// TIA Portal V16 export
// export: Created 2022-11-17T11:55:05.4480097Z, ExportSetting WithDefaults, DisplayName Totally Integrated Automation Portal, DisplayVersion V16 Update 6, DisplayName TIA Portal Version Control Interface, DisplayVersion V16 Update 2, DisplayName TIA Portal Openness, DisplayVersion V16 Update 6, DisplayName SINAMICS Startdrive Advanced, DisplayVersion V16 Update 5, DisplayName SINAMICS Startdrive G130, G150, S120, S150, SINAMICS MV, S210, DisplayVersion V16 Update 5, DisplayName SINAMICS Startdrive G110M, G120, G120C, G120D, G120P, G115D, DisplayVersion V16 Update 5, DisplayName STEP 7 Professional, DisplayVersion V16 Update 6, DisplayName STEP 7 Safety, DisplayVersion V16, DisplayName WinCC Advanced, DisplayVersion V16 Update 6
FUNCTION "FC08_SpoolCarriagePos" : Void   // FC8, LAD
TITLE = Spool carriages Helix40/2 positioning
{ S7_Optimized_Access := 'FALSE' }
AUTHOR : Robopac
VERSION : 0.0
// stored: AutoNumber false, IsIECCheckEnabled false, SetENOAutomatically false, UDAEnableTagReadback false
   VAR_TEMP
      Isteresi : Int;
      TempInt : Int;
      Encoder : Int;
      TempDint1 : DInt;
      TempWord : Word;
      TempDint2 : DInt;
   END_VAR
   VAR_TEMP   // added for the SCL form of the ladder/FBD networks
      _w1 : Bool;
      _w2 : Bool;
   END_VAR
BEGIN

REGION Network 1: Reset spool carriage positioning counter (pulse)
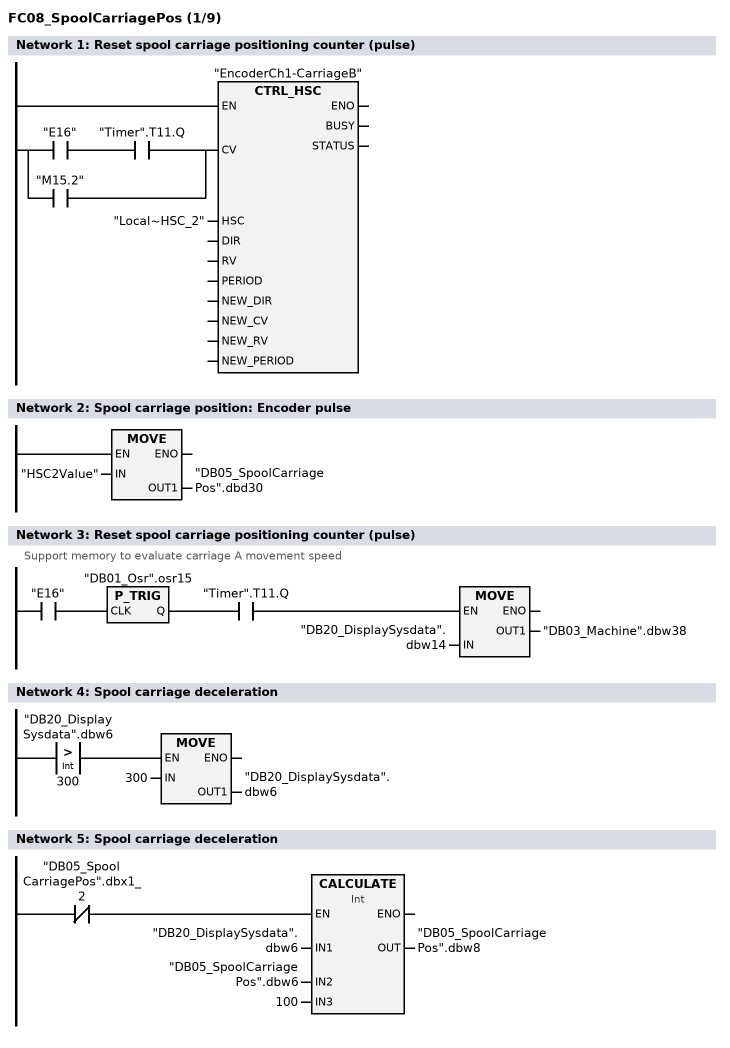
   RUNG wire#powerrail
      "EncoderCh1-CarriageB".CTRL_HSC(CV := wire#w1, HSC := "Local~HSC_2", DIR :=, RV :=, PERIOD :=, NEW_DIR :=, NEW_CV :=, NEW_RV :=, NEW_PERIOD :=, BUSY =>, STATUS =>)
   END_RUNG
   RUNG wire#powerrail
      Contact( "E16" )
      Contact( "Timer".T11.Q )
   END_RUNG wire#w1
   RUNG wire#powerrail
      Contact( "M15.2" )
   END_RUNG wire#w1
   // the same network as SCL:
   "EncoderCh1-CarriageB"(CV := ("E16" AND "Timer".T11.Q) OR "M15.2", HSC := "Local~HSC_2");   // CTRL_HSC
END_REGION

REGION Network 2: Spool carriage position: Encoder pulse
   RUNG wire#powerrail
      { S7_GenerateENO := "TRUE" } Move(in := "HSC2Value", out1 => "DB05_SpoolCarriagePos".dbd30)
   END_RUNG
   // the same network as SCL:
   "DB05_SpoolCarriagePos".dbd30 := "HSC2Value";
END_REGION

REGION Network 3: Reset spool carriage positioning counter (pulse)
   // Support memory to evaluate carriage A movement speed
   RUNG wire#powerrail
      Contact( "E16" )
      P_Trig( "DB01_Osr".osr15 )
      Contact( "Timer".T11.Q )
      { S7_GenerateENO := "TRUE" } Move(in := "DB20_DisplaySysdata".dbw14, out1 => "DB03_Machine".dbw38)
   END_RUNG
   // the same network as SCL:
   #_w1 := "E16" AND NOT "DB01_Osr".osr15;   // rising edge
   "DB01_Osr".osr15 := "E16";
   IF #_w1 AND "Timer".T11.Q THEN "DB03_Machine".dbw38 := "DB20_DisplaySysdata".dbw14; END_IF;
END_REGION

REGION Network 4: Spool carriage deceleration
   RUNG wire#powerrail
      { S7_Templates := "SrcType := Int" } GT_Contact(in1 := "DB20_DisplaySysdata".dbw6, in2 := 300)
      { S7_GenerateENO := "TRUE" } Move(in := 300, out1 => "DB20_DisplaySysdata".dbw6)
   END_RUNG
   // the same network as SCL:
   IF "DB20_DisplaySysdata".dbw6 > 300 THEN "DB20_DisplaySysdata".dbw6 := 300; END_IF;
END_REGION

REGION Network 5: Spool carriage deceleration
   RUNG wire#powerrail
      I_Contact( "DB05_SpoolCarriagePos".dbx1_2 )
      { S7_Templates := "SrcType := Int"; S7_GenerateENO := "TRUE"; S7_Expression := "In1 * In2 / In3" } Calculate(in1 := "DB20_DisplaySysdata".dbw6, in2 := "DB05_SpoolCarriagePos".dbw6, in3 := 100, out => "DB05_SpoolCarriagePos".dbw8)
   END_RUNG
   // the same network as SCL:
   IF NOT "DB05_SpoolCarriagePos".dbx1_2 THEN
       "DB05_SpoolCarriagePos".dbw8 := "DB20_DisplaySysdata".dbw6 * "DB05_SpoolCarriagePos".dbw6 / 100;
   END_IF;
END_REGION

REGION Network 6: Spool carriage position and deceleration
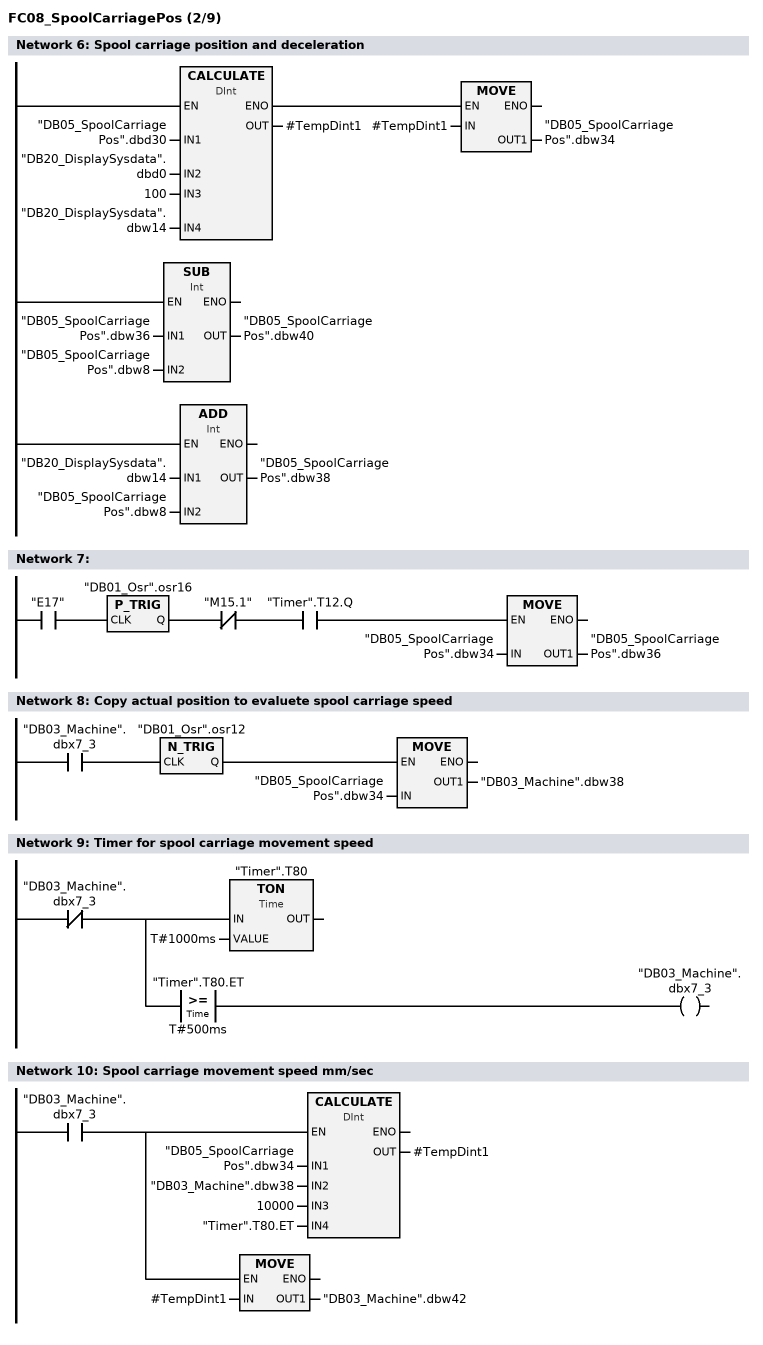
   RUNG wire#powerrail
      { S7_Templates := "SrcType := DInt"; S7_GenerateENO := "TRUE"; S7_Expression := "((In1*In2)/In3)+In4" } Calculate(in1 := "DB05_SpoolCarriagePos".dbd30, in2 := "DB20_DisplaySysdata".dbd0, in3 := 100, in4 := "DB20_DisplaySysdata".dbw14, out => #TempDint1)
      { S7_GenerateENO := "TRUE" } Move(in := #TempDint1, out1 => "DB05_SpoolCarriagePos".dbw34)
   END_RUNG
   RUNG wire#powerrail
      { S7_Templates := "SrcType := Int"; S7_GenerateENO := "TRUE" } Sub(in1 := "DB05_SpoolCarriagePos".dbw36, in2 := "DB05_SpoolCarriagePos".dbw8, out => "DB05_SpoolCarriagePos".dbw40)
   END_RUNG
   RUNG wire#powerrail
      { S7_Templates := "SrcType := Int"; S7_GenerateENO := "TRUE" } Add(in1 := "DB20_DisplaySysdata".dbw14, in2 := "DB05_SpoolCarriagePos".dbw8, out => "DB05_SpoolCarriagePos".dbw38)
   END_RUNG
   // the same network as SCL:
   // ENO of a box is taken as its EN; it also drops when the box reports an error
   #TempDint1 := (("DB05_SpoolCarriagePos".dbd30*"DB20_DisplaySysdata".dbd0)/100)+"DB20_DisplaySysdata".dbw14;
   "DB05_SpoolCarriagePos".dbw34 := #TempDint1;
   "DB05_SpoolCarriagePos".dbw40 := "DB05_SpoolCarriagePos".dbw36 - "DB05_SpoolCarriagePos".dbw8;
   "DB05_SpoolCarriagePos".dbw38 := "DB20_DisplaySysdata".dbw14 + "DB05_SpoolCarriagePos".dbw8;
END_REGION

REGION Network 7
   RUNG wire#powerrail
      Contact( "E17" )
      P_Trig( "DB01_Osr".osr16 )
      I_Contact( "M15.1" )
      Contact( "Timer".T12.Q )
      { S7_GenerateENO := "TRUE" } Move(in := "DB05_SpoolCarriagePos".dbw34, out1 => "DB05_SpoolCarriagePos".dbw36)
   END_RUNG
   // the same network as SCL:
   #_w1 := "E17" AND NOT "DB01_Osr".osr16;   // rising edge
   "DB01_Osr".osr16 := "E17";
   IF #_w1 AND NOT "M15.1" AND "Timer".T12.Q THEN
       "DB05_SpoolCarriagePos".dbw36 := "DB05_SpoolCarriagePos".dbw34;
   END_IF;
END_REGION

REGION Network 8: Copy actual position to evaluete spool carriage speed
   RUNG wire#powerrail
      Contact( "DB03_Machine".dbx7_3 )
      N_Trig( "DB01_Osr".osr12 )
      { S7_GenerateENO := "TRUE" } Move(in := "DB05_SpoolCarriagePos".dbw34, out1 => "DB03_Machine".dbw38)
   END_RUNG
   // the same network as SCL:
   #_w1 := NOT "DB03_Machine".dbx7_3 AND "DB01_Osr".osr12;   // falling edge
   "DB01_Osr".osr12 := "DB03_Machine".dbx7_3;
   IF #_w1 THEN "DB03_Machine".dbw38 := "DB05_SpoolCarriagePos".dbw34; END_IF;
END_REGION

REGION Network 9: Timer for spool carriage movement speed
   #_w1 := NOT "DB03_Machine".dbx7_3;
   "Timer".T80.TON(IN := #_w1, PT := T#1000ms);   // TON coil
   "DB03_Machine".dbx7_3 := #_w1 AND ("Timer".T80.ET >= T#500ms);
END_REGION

REGION Network 10: Spool carriage movement speed mm/sec
   RUNG wire#powerrail
      Contact( "DB03_Machine".dbx7_3 )
      wire#w1
      { S7_Templates := "SrcType := DInt"; S7_GenerateENO := "TRUE"; S7_Expression := "(In1-In2)*In3/In4" } Calculate(in1 := "DB05_SpoolCarriagePos".dbw34, in2 := "DB03_Machine".dbw38, in3 := 10000, in4 := "Timer".T80.ET, out => #TempDint1)
   END_RUNG
   RUNG wire#w1
      { S7_GenerateENO := "TRUE" } Move(in := #TempDint1, out1 => "DB03_Machine".dbw42)
   END_RUNG
   // the same network as SCL:
   IF "DB03_Machine".dbx7_3 THEN
       #TempDint1 := ("DB05_SpoolCarriagePos".dbw34-"DB03_Machine".dbw38)*10000/"Timer".T80.ET;
       "DB03_Machine".dbw42 := #TempDint1;
   END_IF;
END_REGION

REGION Network 11: Spool carriage movement speed mm/sec recorded
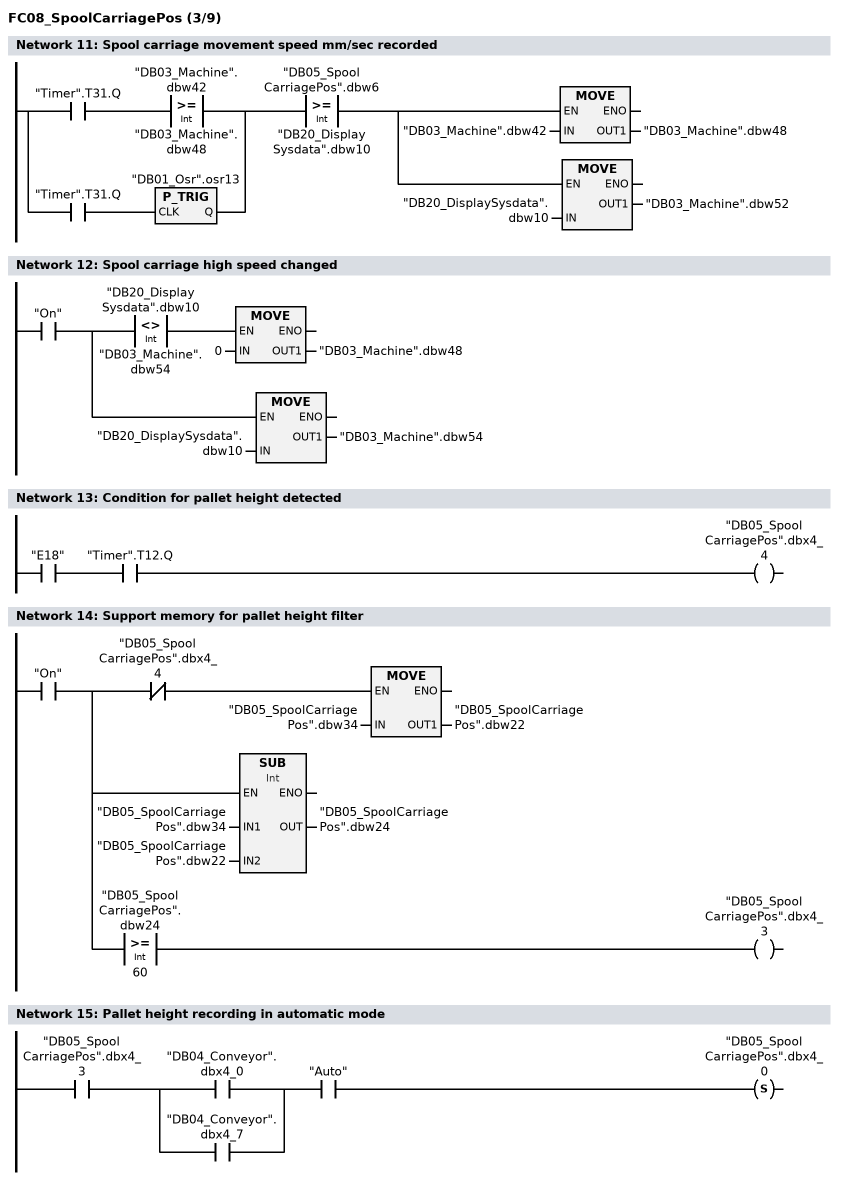
   RUNG wire#powerrail
      Contact( "Timer".T31.Q )
      { S7_Templates := "SrcType := Int" } GE_Contact(in1 := "DB03_Machine".dbw42, in2 := "DB03_Machine".dbw48)
      wire#w1
      { S7_Templates := "SrcType := Int" } GE_Contact(in1 := "DB05_SpoolCarriagePos".dbw6, in2 := "DB20_DisplaySysdata".dbw10)
      wire#w2
      { S7_GenerateENO := "TRUE" } Move(in := "DB03_Machine".dbw42, out1 => "DB03_Machine".dbw48)
   END_RUNG
   RUNG wire#powerrail
      Contact( "Timer".T31.Q )
      P_Trig( "DB01_Osr".osr13 )
   END_RUNG wire#w1
   RUNG wire#w2
      { S7_GenerateENO := "TRUE" } Move(in := "DB20_DisplaySysdata".dbw10, out1 => "DB03_Machine".dbw52)
   END_RUNG
   // the same network as SCL:
   #_w1 := "Timer".T31.Q AND NOT "DB01_Osr".osr13;   // rising edge
   "DB01_Osr".osr13 := "Timer".T31.Q;
   #_w2 := (("Timer".T31.Q AND ("DB03_Machine".dbw42 >= "DB03_Machine".dbw48)) OR #_w1) AND ("DB05_SpoolCarriagePos".dbw6 >= "DB20_DisplaySysdata".dbw10);
   IF #_w2 THEN
       "DB03_Machine".dbw48 := "DB03_Machine".dbw42;
       "DB03_Machine".dbw52 := "DB20_DisplaySysdata".dbw10;
   END_IF;
END_REGION

REGION Network 12: Spool carriage high speed changed
   RUNG wire#powerrail
      Contact( "On" )
      wire#w1
      { S7_Templates := "SrcType := Int" } NE_Contact(in1 := "DB20_DisplaySysdata".dbw10, in2 := "DB03_Machine".dbw54)
      { S7_GenerateENO := "TRUE" } Move(in := 0, out1 => "DB03_Machine".dbw48)
   END_RUNG
   RUNG wire#w1
      { S7_GenerateENO := "TRUE" } Move(in := "DB20_DisplaySysdata".dbw10, out1 => "DB03_Machine".dbw54)
   END_RUNG
   // the same network as SCL:
   IF "On" AND ("DB20_DisplaySysdata".dbw10 <> "DB03_Machine".dbw54) THEN "DB03_Machine".dbw48 := 0; END_IF;
   IF "On" THEN "DB03_Machine".dbw54 := "DB20_DisplaySysdata".dbw10; END_IF;
END_REGION

REGION Network 13: Condition for pallet height detected
   RUNG wire#powerrail
      Contact( "E18" )
      Contact( "Timer".T12.Q )
      Coil( "DB05_SpoolCarriagePos".dbx4_4 )
   END_RUNG
   // the same network as SCL:
   "DB05_SpoolCarriagePos".dbx4_4 := "E18" AND "Timer".T12.Q;
END_REGION

REGION Network 14: Support memory for pallet height filter
   RUNG wire#powerrail
      Contact( "On" )
      wire#w1
      I_Contact( "DB05_SpoolCarriagePos".dbx4_4 )
      { S7_GenerateENO := "TRUE" } Move(in := "DB05_SpoolCarriagePos".dbw34, out1 => "DB05_SpoolCarriagePos".dbw22)
   END_RUNG
   RUNG wire#w1
      { S7_Templates := "SrcType := Int"; S7_GenerateENO := "TRUE" } Sub(in1 := "DB05_SpoolCarriagePos".dbw34, in2 := "DB05_SpoolCarriagePos".dbw22, out => "DB05_SpoolCarriagePos".dbw24)
   END_RUNG
   RUNG wire#w1
      { S7_Templates := "SrcType := Int" } GE_Contact(in1 := "DB05_SpoolCarriagePos".dbw24, in2 := 60)
      Coil( "DB05_SpoolCarriagePos".dbx4_3 )
   END_RUNG
   // the same network as SCL:
   IF "On" AND NOT "DB05_SpoolCarriagePos".dbx4_4 THEN
       "DB05_SpoolCarriagePos".dbw22 := "DB05_SpoolCarriagePos".dbw34;
   END_IF;
   IF "On" THEN
       "DB05_SpoolCarriagePos".dbw24 := "DB05_SpoolCarriagePos".dbw34 - "DB05_SpoolCarriagePos".dbw22;
   END_IF;
   "DB05_SpoolCarriagePos".dbx4_3 := "On" AND ("DB05_SpoolCarriagePos".dbw24 >= 60);
END_REGION

REGION Network 15: Pallet height recording in automatic mode
   RUNG wire#powerrail
      Contact( "DB05_SpoolCarriagePos".dbx4_3 )
      wire#w1
      Contact( "DB04_Conveyor".dbx4_0 )
      wire#w2
      Contact( "Auto" )
      S_Coil( "DB05_SpoolCarriagePos".dbx4_0 )
   END_RUNG
   RUNG wire#w1
      Contact( "DB04_Conveyor".dbx4_7 )
   END_RUNG wire#w2
   // the same network as SCL:
   IF "DB05_SpoolCarriagePos".dbx4_3 AND ("DB04_Conveyor".dbx4_0 OR "DB04_Conveyor".dbx4_7) AND "Auto" THEN
       "DB05_SpoolCarriagePos".dbx4_0 := TRUE;
   END_IF;
END_REGION

REGION Network 16: Recording pallet height for wrapping position
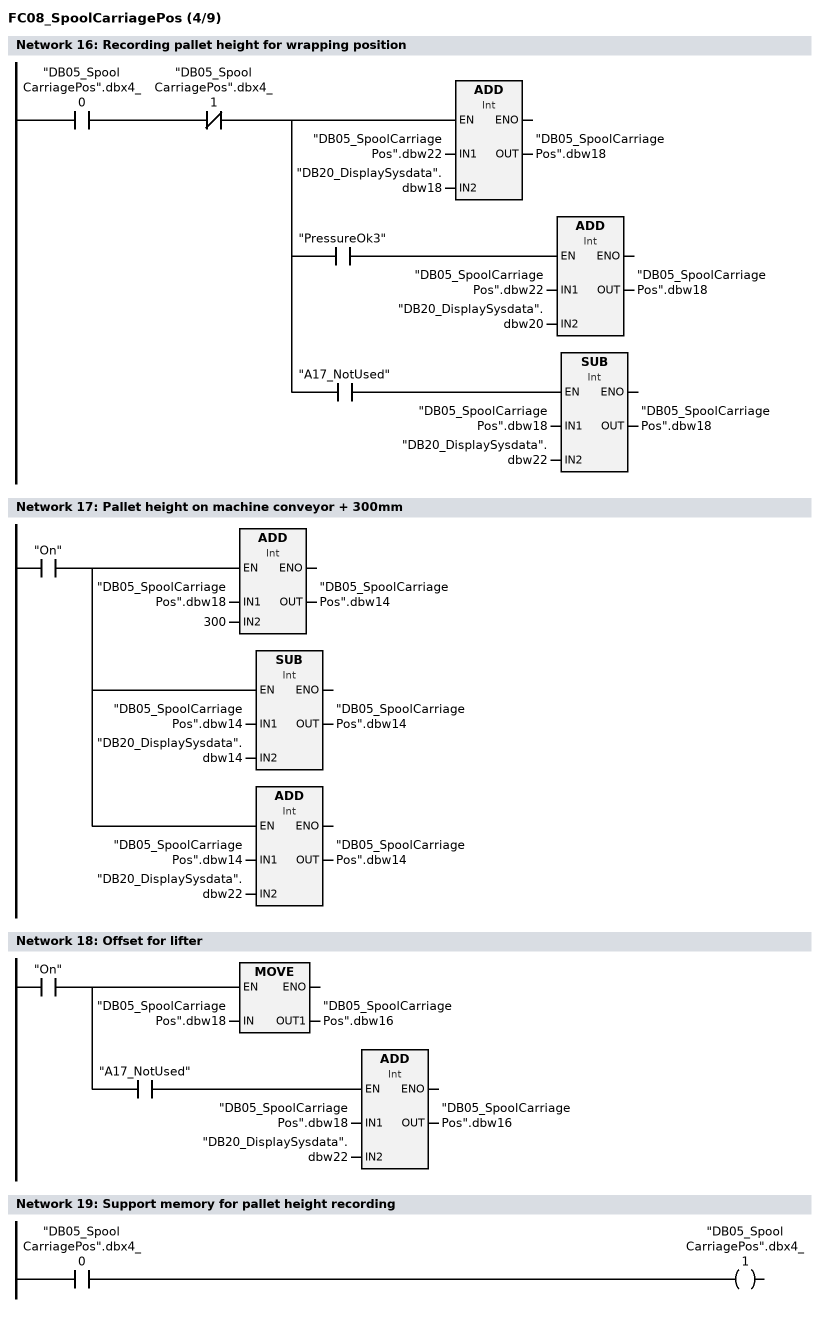
   RUNG wire#powerrail
      Contact( "DB05_SpoolCarriagePos".dbx4_0 )
      I_Contact( "DB05_SpoolCarriagePos".dbx4_1 )
      wire#w1
      { S7_Templates := "SrcType := Int"; S7_GenerateENO := "TRUE" } Add(in1 := "DB05_SpoolCarriagePos".dbw22, in2 := "DB20_DisplaySysdata".dbw18, out => "DB05_SpoolCarriagePos".dbw18)
   END_RUNG
   RUNG wire#w1
      Contact( "PressureOk3" )
      { S7_Templates := "SrcType := Int"; S7_GenerateENO := "TRUE" } Add(in1 := "DB05_SpoolCarriagePos".dbw22, in2 := "DB20_DisplaySysdata".dbw20, out => "DB05_SpoolCarriagePos".dbw18)
   END_RUNG
   RUNG wire#w1
      Contact( "A17_NotUsed" )
      { S7_Templates := "SrcType := Int"; S7_GenerateENO := "TRUE" } Sub(in1 := "DB05_SpoolCarriagePos".dbw18, in2 := "DB20_DisplaySysdata".dbw22, out => "DB05_SpoolCarriagePos".dbw18)
   END_RUNG
   // the same network as SCL:
   #_w1 := "DB05_SpoolCarriagePos".dbx4_0 AND NOT "DB05_SpoolCarriagePos".dbx4_1;
   IF #_w1 THEN
       "DB05_SpoolCarriagePos".dbw18 := "DB05_SpoolCarriagePos".dbw22 + "DB20_DisplaySysdata".dbw18;
   END_IF;
   IF #_w1 AND "PressureOk3" THEN
       "DB05_SpoolCarriagePos".dbw18 := "DB05_SpoolCarriagePos".dbw22 + "DB20_DisplaySysdata".dbw20;
   END_IF;
   IF #_w1 AND "A17_NotUsed" THEN
       "DB05_SpoolCarriagePos".dbw18 := "DB05_SpoolCarriagePos".dbw18 - "DB20_DisplaySysdata".dbw22;
   END_IF;
END_REGION

REGION Network 17: Pallet height on machine conveyor + 300mm
   RUNG wire#powerrail
      Contact( "On" )
      wire#w1
      { S7_Templates := "SrcType := Int"; S7_GenerateENO := "TRUE" } Add(in1 := "DB05_SpoolCarriagePos".dbw18, in2 := 300, out => "DB05_SpoolCarriagePos".dbw14)
   END_RUNG
   RUNG wire#w1
      { S7_Templates := "SrcType := Int"; S7_GenerateENO := "TRUE" } Sub(in1 := "DB05_SpoolCarriagePos".dbw14, in2 := "DB20_DisplaySysdata".dbw14, out => "DB05_SpoolCarriagePos".dbw14)
   END_RUNG
   RUNG wire#w1
      { S7_Templates := "SrcType := Int"; S7_GenerateENO := "TRUE" } Add(in1 := "DB05_SpoolCarriagePos".dbw14, in2 := "DB20_DisplaySysdata".dbw22, out => "DB05_SpoolCarriagePos".dbw14)
   END_RUNG
   // the same network as SCL:
   IF "On" THEN
       "DB05_SpoolCarriagePos".dbw14 := "DB05_SpoolCarriagePos".dbw18 + 300;
       "DB05_SpoolCarriagePos".dbw14 := "DB05_SpoolCarriagePos".dbw14 - "DB20_DisplaySysdata".dbw14;
       "DB05_SpoolCarriagePos".dbw14 := "DB05_SpoolCarriagePos".dbw14 + "DB20_DisplaySysdata".dbw22;
   END_IF;
END_REGION

REGION Network 18: Offset for lifter
   RUNG wire#powerrail
      Contact( "On" )
      wire#w1
      { S7_GenerateENO := "TRUE" } Move(in := "DB05_SpoolCarriagePos".dbw18, out1 => "DB05_SpoolCarriagePos".dbw16)
   END_RUNG
   RUNG wire#w1
      Contact( "A17_NotUsed" )
      { S7_Templates := "SrcType := Int"; S7_GenerateENO := "TRUE" } Add(in1 := "DB05_SpoolCarriagePos".dbw18, in2 := "DB20_DisplaySysdata".dbw22, out => "DB05_SpoolCarriagePos".dbw16)
   END_RUNG
   // the same network as SCL:
   IF "On" THEN "DB05_SpoolCarriagePos".dbw16 := "DB05_SpoolCarriagePos".dbw18; END_IF;
   IF "On" AND "A17_NotUsed" THEN
       "DB05_SpoolCarriagePos".dbw16 := "DB05_SpoolCarriagePos".dbw18 + "DB20_DisplaySysdata".dbw22;
   END_IF;
END_REGION

REGION Network 19: Support memory for pallet height recording
   RUNG wire#powerrail
      Contact( "DB05_SpoolCarriagePos".dbx4_0 )
      Coil( "DB05_SpoolCarriagePos".dbx4_1 )
   END_RUNG
   // the same network as SCL:
   "DB05_SpoolCarriagePos".dbx4_1 := "DB05_SpoolCarriagePos".dbx4_0;
END_REGION

REGION Network 20: Pallet height recording in automatic mode
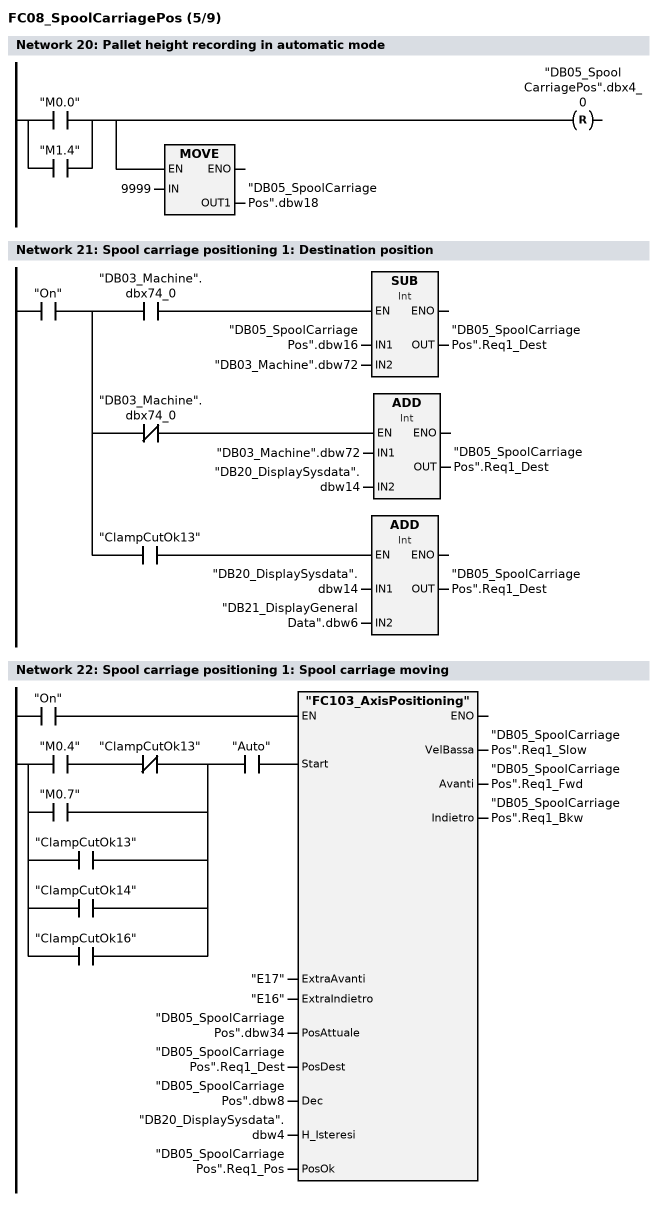
   RUNG wire#powerrail
      Contact( "M0.0" )
      wire#w1
      R_Coil( "DB05_SpoolCarriagePos".dbx4_0 )
   END_RUNG
   RUNG wire#powerrail
      Contact( "M1.4" )
   END_RUNG wire#w1
   RUNG wire#w1
      { S7_GenerateENO := "TRUE" } Move(in := 9999, out1 => "DB05_SpoolCarriagePos".dbw18)
   END_RUNG
   // the same network as SCL:
   IF "M0.0" OR "M1.4" THEN
       "DB05_SpoolCarriagePos".dbx4_0 := FALSE;
       "DB05_SpoolCarriagePos".dbw18 := 9999;
   END_IF;
END_REGION

REGION Network 21: Spool carriage positioning 1: Destination position
   RUNG wire#powerrail
      Contact( "On" )
      wire#w1
      Contact( "DB03_Machine".dbx74_0 )
      { S7_Templates := "SrcType := Int"; S7_GenerateENO := "TRUE" } Sub(in1 := "DB05_SpoolCarriagePos".dbw16, in2 := "DB03_Machine".dbw72, out => "DB05_SpoolCarriagePos".Req1_Dest)
   END_RUNG
   RUNG wire#w1
      I_Contact( "DB03_Machine".dbx74_0 )
      { S7_Templates := "SrcType := Int"; S7_GenerateENO := "TRUE" } Add(in1 := "DB03_Machine".dbw72, in2 := "DB20_DisplaySysdata".dbw14, out => "DB05_SpoolCarriagePos".Req1_Dest)
   END_RUNG
   RUNG wire#w1
      Contact( "ClampCutOk13" )
      { S7_Templates := "SrcType := Int"; S7_GenerateENO := "TRUE" } Add(in1 := "DB20_DisplaySysdata".dbw14, in2 := "DB21_DisplayGeneralData".dbw6, out => "DB05_SpoolCarriagePos".Req1_Dest)
   END_RUNG
   // the same network as SCL:
   IF "On" AND "DB03_Machine".dbx74_0 THEN
       "DB05_SpoolCarriagePos".Req1_Dest := "DB05_SpoolCarriagePos".dbw16 - "DB03_Machine".dbw72;
   END_IF;
   IF "On" AND NOT "DB03_Machine".dbx74_0 THEN
       "DB05_SpoolCarriagePos".Req1_Dest := "DB03_Machine".dbw72 + "DB20_DisplaySysdata".dbw14;
   END_IF;
   IF "On" AND "ClampCutOk13" THEN
       "DB05_SpoolCarriagePos".Req1_Dest := "DB20_DisplaySysdata".dbw14 + "DB21_DisplayGeneralData".dbw6;
   END_IF;
END_REGION

REGION Network 22: Spool carriage positioning 1: Spool carriage moving
   RUNG wire#powerrail
      Contact( "On" )
      "FC103_AxisPositioning"(Start := wire#w2, ExtraAvanti := "E17", ExtraIndietro := "E16", PosAttuale := "DB05_SpoolCarriagePos".dbw34, PosDest := "DB05_SpoolCarriagePos".Req1_Dest, Dec := "DB05_SpoolCarriagePos".dbw8, H_Isteresi := "DB20_DisplaySysdata".dbw4, PosOk := "DB05_SpoolCarriagePos".Req1_Pos, VelBassa => "DB05_SpoolCarriagePos".Req1_Slow, Avanti => "DB05_SpoolCarriagePos".Req1_Fwd, Indietro => "DB05_SpoolCarriagePos".Req1_Bkw)
   END_RUNG
   RUNG wire#powerrail
      Contact( "M0.4" )
      I_Contact( "ClampCutOk13" )
      wire#w1
      Contact( "Auto" )
   END_RUNG wire#w2
   RUNG wire#powerrail
      Contact( "M0.7" )
   END_RUNG wire#w1
   RUNG wire#powerrail
      Contact( "ClampCutOk13" )
   END_RUNG wire#w1
   RUNG wire#powerrail
      Contact( "ClampCutOk14" )
   END_RUNG wire#w1
   RUNG wire#powerrail
      Contact( "ClampCutOk16" )
   END_RUNG wire#w1
   // the same network as SCL:
   IF "On" THEN
       "FC103_AxisPositioning"(Start := (("M0.4" AND NOT "ClampCutOk13") OR "M0.7" OR "ClampCutOk13" OR "ClampCutOk14" OR "ClampCutOk16") AND "Auto",
                               ExtraAvanti := "E17",
                               ExtraIndietro := "E16",
                               PosAttuale := "DB05_SpoolCarriagePos".dbw34,
                               PosDest := "DB05_SpoolCarriagePos".Req1_Dest,
                               Dec := "DB05_SpoolCarriagePos".dbw8,
                               H_Isteresi := "DB20_DisplaySysdata".dbw4,
                               PosOk := "DB05_SpoolCarriagePos".Req1_Pos,
                               VelBassa => "DB05_SpoolCarriagePos".Req1_Slow,
                               Avanti => "DB05_SpoolCarriagePos".Req1_Fwd,
                               Indietro => "DB05_SpoolCarriagePos".Req1_Bkw);
   END_IF;
END_REGION

REGION Network 23: Spool carriage positioning 2: Destination position
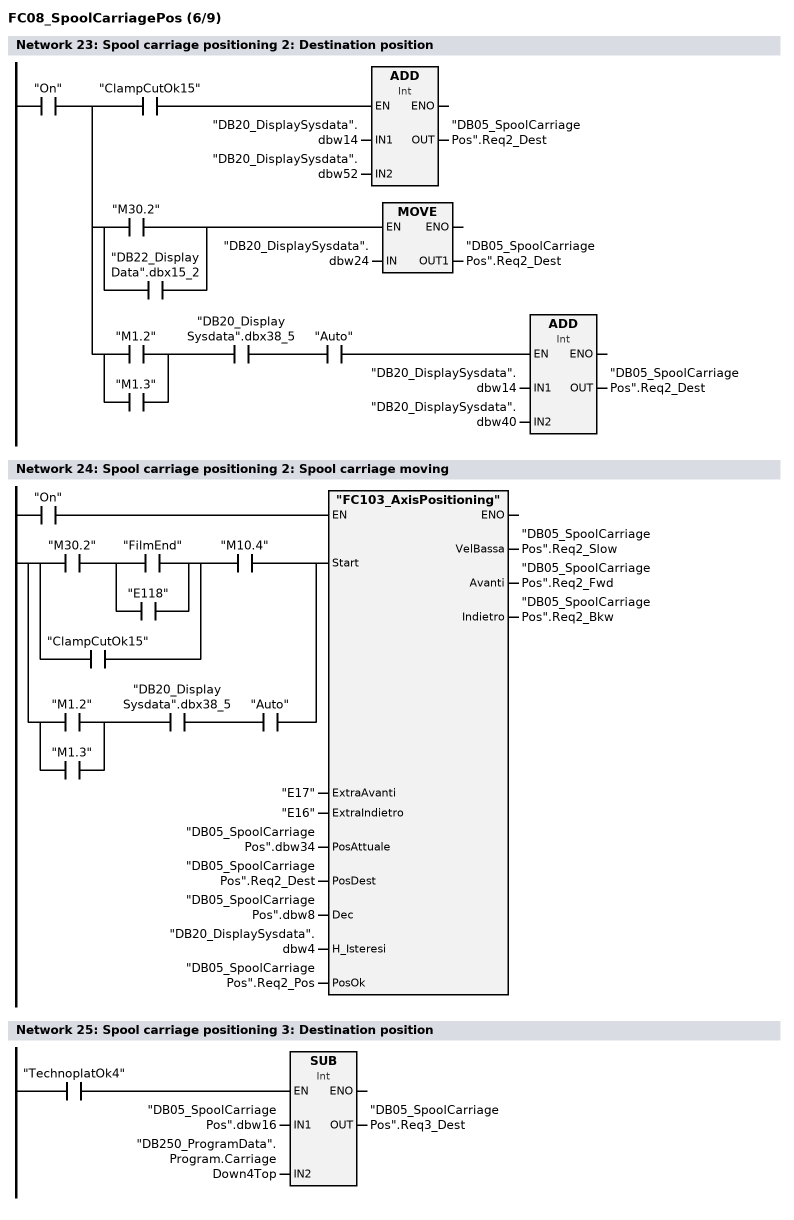
   RUNG wire#powerrail
      Contact( "On" )
      wire#w1
      Contact( "ClampCutOk15" )
      { S7_Templates := "SrcType := Int"; S7_GenerateENO := "TRUE" } Add(in1 := "DB20_DisplaySysdata".dbw14, in2 := "DB20_DisplaySysdata".dbw52, out => "DB05_SpoolCarriagePos".Req2_Dest)
   END_RUNG
   RUNG wire#w1
      Contact( "M30.2" )
      wire#w2
      { S7_GenerateENO := "TRUE" } Move(in := "DB20_DisplaySysdata".dbw24, out1 => "DB05_SpoolCarriagePos".Req2_Dest)
   END_RUNG
   RUNG wire#w1
      Contact( "DB22_DisplayData".dbx15_2 )
   END_RUNG wire#w2
   RUNG wire#w1
      Contact( "M1.2" )
      wire#w3
      Contact( "DB20_DisplaySysdata".dbx38_5 )
      Contact( "Auto" )
      { S7_Templates := "SrcType := Int"; S7_GenerateENO := "TRUE" } Add(in1 := "DB20_DisplaySysdata".dbw14, in2 := "DB20_DisplaySysdata".dbw40, out => "DB05_SpoolCarriagePos".Req2_Dest)
   END_RUNG
   RUNG wire#w1
      Contact( "M1.3" )
   END_RUNG wire#w3
   // the same network as SCL:
   IF "On" AND "ClampCutOk15" THEN
       "DB05_SpoolCarriagePos".Req2_Dest := "DB20_DisplaySysdata".dbw14 + "DB20_DisplaySysdata".dbw52;
   END_IF;
   IF "On" AND ("M30.2" OR "DB22_DisplayData".dbx15_2) THEN
       "DB05_SpoolCarriagePos".Req2_Dest := "DB20_DisplaySysdata".dbw24;
   END_IF;
   IF "On" AND ("M1.2" OR "M1.3") AND "DB20_DisplaySysdata".dbx38_5 AND "Auto" THEN
       "DB05_SpoolCarriagePos".Req2_Dest := "DB20_DisplaySysdata".dbw14 + "DB20_DisplaySysdata".dbw40;
   END_IF;
END_REGION

REGION Network 24: Spool carriage positioning 2: Spool carriage moving
   RUNG wire#powerrail
      Contact( "On" )
      "FC103_AxisPositioning"(Start := wire#w4, ExtraAvanti := "E17", ExtraIndietro := "E16", PosAttuale := "DB05_SpoolCarriagePos".dbw34, PosDest := "DB05_SpoolCarriagePos".Req2_Dest, Dec := "DB05_SpoolCarriagePos".dbw8, H_Isteresi := "DB20_DisplaySysdata".dbw4, PosOk := "DB05_SpoolCarriagePos".Req2_Pos, VelBassa => "DB05_SpoolCarriagePos".Req2_Slow, Avanti => "DB05_SpoolCarriagePos".Req2_Fwd, Indietro => "DB05_SpoolCarriagePos".Req2_Bkw)
   END_RUNG
   RUNG wire#powerrail
      Contact( "M30.2" )
      wire#w1
      Contact( "FilmEnd" )
      wire#w2
      Contact( "M10.4" )
   END_RUNG wire#w4
   RUNG wire#w1
      Contact( "E118" )
   END_RUNG wire#w2
   RUNG wire#powerrail
      Contact( "ClampCutOk15" )
   END_RUNG wire#w2
   RUNG wire#powerrail
      Contact( "M1.2" )
      wire#w3
      Contact( "DB20_DisplaySysdata".dbx38_5 )
      Contact( "Auto" )
   END_RUNG wire#w4
   RUNG wire#powerrail
      Contact( "M1.3" )
   END_RUNG wire#w3
   // the same network as SCL:
   IF "On" THEN
       "FC103_AxisPositioning"(Start := ((("M30.2" AND ("FilmEnd" OR "E118")) OR "ClampCutOk15") AND "M10.4") OR (("M1.2" OR "M1.3") AND "DB20_DisplaySysdata".dbx38_5 AND "Auto"),
                               ExtraAvanti := "E17",
                               ExtraIndietro := "E16",
                               PosAttuale := "DB05_SpoolCarriagePos".dbw34,
                               PosDest := "DB05_SpoolCarriagePos".Req2_Dest,
                               Dec := "DB05_SpoolCarriagePos".dbw8,
                               H_Isteresi := "DB20_DisplaySysdata".dbw4,
                               PosOk := "DB05_SpoolCarriagePos".Req2_Pos,
                               VelBassa => "DB05_SpoolCarriagePos".Req2_Slow,
                               Avanti => "DB05_SpoolCarriagePos".Req2_Fwd,
                               Indietro => "DB05_SpoolCarriagePos".Req2_Bkw);
   END_IF;
END_REGION

REGION Network 25: Spool carriage positioning 3: Destination position
   RUNG wire#powerrail
      Contact( "TechnoplatOk4" )
      { S7_Templates := "SrcType := Int"; S7_GenerateENO := "TRUE" } Sub(in1 := "DB05_SpoolCarriagePos".dbw16, in2 := "DB250_ProgramData".Program.CarriageDown4Top, out => "DB05_SpoolCarriagePos".Req3_Dest)
   END_RUNG
   // the same network as SCL:
   IF "TechnoplatOk4" THEN
       "DB05_SpoolCarriagePos".Req3_Dest := "DB05_SpoolCarriagePos".dbw16 - "DB250_ProgramData".Program.CarriageDown4Top;
   END_IF;
END_REGION

REGION Network 26: Spool carriage positioning 3: Spool carriage moving
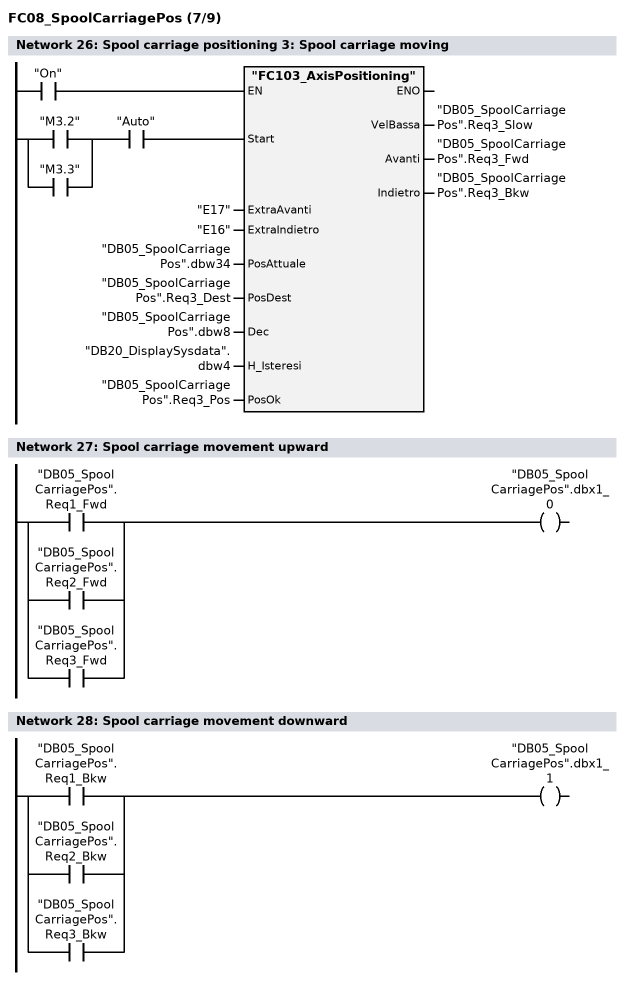
   RUNG wire#powerrail
      Contact( "On" )
      "FC103_AxisPositioning"(Start := wire#w2, ExtraAvanti := "E17", ExtraIndietro := "E16", PosAttuale := "DB05_SpoolCarriagePos".dbw34, PosDest := "DB05_SpoolCarriagePos".Req3_Dest, Dec := "DB05_SpoolCarriagePos".dbw8, H_Isteresi := "DB20_DisplaySysdata".dbw4, PosOk := "DB05_SpoolCarriagePos".Req3_Pos, VelBassa => "DB05_SpoolCarriagePos".Req3_Slow, Avanti => "DB05_SpoolCarriagePos".Req3_Fwd, Indietro => "DB05_SpoolCarriagePos".Req3_Bkw)
   END_RUNG
   RUNG wire#powerrail
      Contact( "M3.2" )
      wire#w1
      Contact( "Auto" )
   END_RUNG wire#w2
   RUNG wire#powerrail
      Contact( "M3.3" )
   END_RUNG wire#w1
   // the same network as SCL:
   IF "On" THEN
       "FC103_AxisPositioning"(Start := ("M3.2" OR "M3.3") AND "Auto",
                               ExtraAvanti := "E17",
                               ExtraIndietro := "E16",
                               PosAttuale := "DB05_SpoolCarriagePos".dbw34,
                               PosDest := "DB05_SpoolCarriagePos".Req3_Dest,
                               Dec := "DB05_SpoolCarriagePos".dbw8,
                               H_Isteresi := "DB20_DisplaySysdata".dbw4,
                               PosOk := "DB05_SpoolCarriagePos".Req3_Pos,
                               VelBassa => "DB05_SpoolCarriagePos".Req3_Slow,
                               Avanti => "DB05_SpoolCarriagePos".Req3_Fwd,
                               Indietro => "DB05_SpoolCarriagePos".Req3_Bkw);
   END_IF;
END_REGION

REGION Network 27: Spool carriage movement upward
   RUNG wire#powerrail
      Contact( "DB05_SpoolCarriagePos".Req1_Fwd )
      wire#w1
      Coil( "DB05_SpoolCarriagePos".dbx1_0 )
   END_RUNG
   RUNG wire#powerrail
      Contact( "DB05_SpoolCarriagePos".Req2_Fwd )
   END_RUNG wire#w1
   RUNG wire#powerrail
      Contact( "DB05_SpoolCarriagePos".Req3_Fwd )
   END_RUNG wire#w1
   // the same network as SCL:
   "DB05_SpoolCarriagePos".dbx1_0 := "DB05_SpoolCarriagePos".Req1_Fwd OR "DB05_SpoolCarriagePos".Req2_Fwd OR "DB05_SpoolCarriagePos".Req3_Fwd;
END_REGION

REGION Network 28: Spool carriage movement downward
   RUNG wire#powerrail
      Contact( "DB05_SpoolCarriagePos".Req1_Bkw )
      wire#w1
      Coil( "DB05_SpoolCarriagePos".dbx1_1 )
   END_RUNG
   RUNG wire#powerrail
      Contact( "DB05_SpoolCarriagePos".Req2_Bkw )
   END_RUNG wire#w1
   RUNG wire#powerrail
      Contact( "DB05_SpoolCarriagePos".Req3_Bkw )
   END_RUNG wire#w1
   // the same network as SCL:
   "DB05_SpoolCarriagePos".dbx1_1 := "DB05_SpoolCarriagePos".Req1_Bkw OR "DB05_SpoolCarriagePos".Req2_Bkw OR "DB05_SpoolCarriagePos".Req3_Bkw;
END_REGION

REGION Network 29: Spool carriage deceleration on carriage positioning
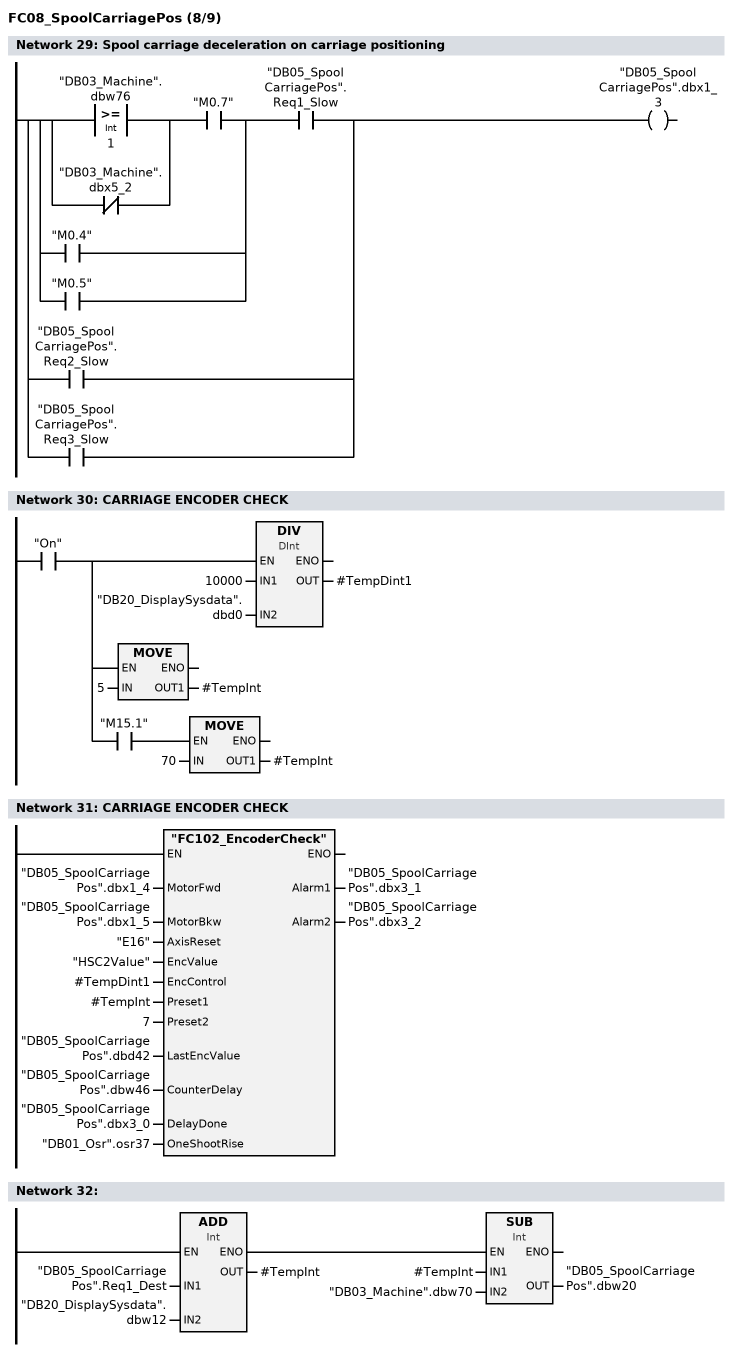
   RUNG wire#powerrail
      { S7_Templates := "SrcType := Int" } GE_Contact(in1 := "DB03_Machine".dbw76, in2 := 1)
      wire#w1
      Contact( "M0.7" )
      wire#w2
      Contact( "DB05_SpoolCarriagePos".Req1_Slow )
      wire#w3
      Coil( "DB05_SpoolCarriagePos".dbx1_3 )
   END_RUNG
   RUNG wire#powerrail
      I_Contact( "DB03_Machine".dbx5_2 )
   END_RUNG wire#w1
   RUNG wire#powerrail
      Contact( "M0.4" )
   END_RUNG wire#w2
   RUNG wire#powerrail
      Contact( "M0.5" )
   END_RUNG wire#w2
   RUNG wire#powerrail
      Contact( "DB05_SpoolCarriagePos".Req2_Slow )
   END_RUNG wire#w3
   RUNG wire#powerrail
      Contact( "DB05_SpoolCarriagePos".Req3_Slow )
   END_RUNG wire#w3
   // the same network as SCL:
   "DB05_SpoolCarriagePos".dbx1_3 := ((((("DB03_Machine".dbw76 >= 1) OR NOT "DB03_Machine".dbx5_2) AND "M0.7") OR "M0.4" OR "M0.5") AND "DB05_SpoolCarriagePos".Req1_Slow) OR "DB05_SpoolCarriagePos".Req2_Slow OR "DB05_SpoolCarriagePos".Req3_Slow;
END_REGION

REGION Network 30: CARRIAGE ENCODER CHECK
   RUNG wire#powerrail
      Contact( "On" )
      wire#w1
      { S7_Templates := "SrcType := DInt"; S7_GenerateENO := "TRUE" } Div(in1 := 10000, in2 := "DB20_DisplaySysdata".dbd0, out => #TempDint1)
   END_RUNG
   RUNG wire#w1
      { S7_GenerateENO := "TRUE" } Move(in := 5, out1 => #TempInt)
   END_RUNG
   RUNG wire#w1
      Contact( "M15.1" )
      { S7_GenerateENO := "TRUE" } Move(in := 70, out1 => #TempInt)
   END_RUNG
   // the same network as SCL:
   IF "On" THEN
       #TempDint1 := 10000 / "DB20_DisplaySysdata".dbd0;
       #TempInt := 5;
   END_IF;
   IF "On" AND "M15.1" THEN #TempInt := 70; END_IF;
END_REGION

REGION Network 31: CARRIAGE ENCODER CHECK
   RUNG wire#powerrail
      "FC102_EncoderCheck"(MotorFwd := "DB05_SpoolCarriagePos".dbx1_4, MotorBkw := "DB05_SpoolCarriagePos".dbx1_5, AxisReset := "E16", EncValue := "HSC2Value", EncControl := #TempDint1, Preset1 := #TempInt, Preset2 := 7, LastEncValue := "DB05_SpoolCarriagePos".dbd42, CounterDelay := "DB05_SpoolCarriagePos".dbw46, DelayDone := "DB05_SpoolCarriagePos".dbx3_0, OneShootRise := "DB01_Osr".osr37, Alarm1 => "DB05_SpoolCarriagePos".dbx3_1, Alarm2 => "DB05_SpoolCarriagePos".dbx3_2)
   END_RUNG
   // the same network as SCL:
   "FC102_EncoderCheck"(MotorFwd := "DB05_SpoolCarriagePos".dbx1_4,
                        MotorBkw := "DB05_SpoolCarriagePos".dbx1_5,
                        AxisReset := "E16",
                        EncValue := "HSC2Value",
                        EncControl := #TempDint1,
                        Preset1 := #TempInt,
                        Preset2 := 7,
                        LastEncValue := "DB05_SpoolCarriagePos".dbd42,
                        CounterDelay := "DB05_SpoolCarriagePos".dbw46,
                        DelayDone := "DB05_SpoolCarriagePos".dbx3_0,
                        OneShootRise := "DB01_Osr".osr37,
                        Alarm1 => "DB05_SpoolCarriagePos".dbx3_1,
                        Alarm2 => "DB05_SpoolCarriagePos".dbx3_2);
END_REGION

REGION Network 32
   RUNG wire#powerrail
      { S7_Templates := "SrcType := Int"; S7_GenerateENO := "TRUE" } Add(in1 := "DB05_SpoolCarriagePos".Req1_Dest, in2 := "DB20_DisplaySysdata".dbw12, out => #TempInt)
      { S7_Templates := "SrcType := Int"; S7_GenerateENO := "TRUE" } Sub(in1 := #TempInt, in2 := "DB03_Machine".dbw70, out => "DB05_SpoolCarriagePos".dbw20)
   END_RUNG
   // the same network as SCL:
   // ENO of a box is taken as its EN; it also drops when the box reports an error
   #TempInt := "DB05_SpoolCarriagePos".Req1_Dest + "DB20_DisplaySysdata".dbw12;
   "DB05_SpoolCarriagePos".dbw20 := #TempInt - "DB03_Machine".dbw70;
END_REGION

REGION Network 33
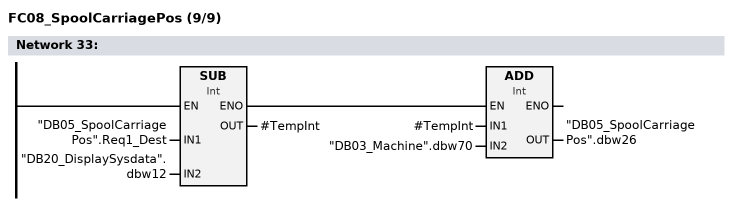
   RUNG wire#powerrail
      { S7_Templates := "SrcType := Int"; S7_GenerateENO := "TRUE" } Sub(in1 := "DB05_SpoolCarriagePos".Req1_Dest, in2 := "DB20_DisplaySysdata".dbw12, out => #TempInt)
      { S7_Templates := "SrcType := Int"; S7_GenerateENO := "TRUE" } Add(in1 := #TempInt, in2 := "DB03_Machine".dbw70, out => "DB05_SpoolCarriagePos".dbw26)
   END_RUNG
   // the same network as SCL:
   // ENO of a box is taken as its EN; it also drops when the box reports an error
   #TempInt := "DB05_SpoolCarriagePos".Req1_Dest - "DB20_DisplaySysdata".dbw12;
   "DB05_SpoolCarriagePos".dbw26 := #TempInt + "DB03_Machine".dbw70;
END_REGION
END_FUNCTION
